Staubli VAL3: Control_ListS.pgx

program Control_ListS(string x_sItemName, num& x_nSelectItem)
  local bool l_bRes
  local string l_sBuff[20]
begin

 call Str_SplitComma(l_bRes,x_sItemName,l_sBuff)
 if !l_bRes
  return
endIf
  call Control_List(l_sBuff,x_nSelectItem)


end
